(* IEC 61131-3 sources: MyReadCfg/sources/MyReadCfg, 2 files *)

(* ---- MyReadCfg.fun ---- *)
{REDUND_ERROR} FUNCTION MRC_Open : UDINT (*Reads a configuration file into memory, returns Ident (0 = error)*) (*$GROUP=User,$CAT=User,$GROUPICON=User.png,$CATICON=User.png*)
	VAR_INPUT
		pDeviceName : UDINT; (*Pointer to FileIO device name, e.g. 'USER' (STRING)*)
		pFileName : UDINT; (*Pointer to file name incl. relative path, e.g. 'Simulation/50000.INI' (STRING)*)
	END_VAR
END_FUNCTION

{REDUND_ERROR} FUNCTION MRC_Close : DINT (*Closes a configuration and frees all resources. 0 = OK*) (*$GROUP=User,$CAT=User,$GROUPICON=User.png,$CATICON=User.png*)
	VAR_INPUT
		Ident : UDINT; (*Ident from MRC_Open*)
	END_VAR
END_FUNCTION

{REDUND_ERROR} FUNCTION MRC_GetLastError : DINT (*Error of the last MyReadCfg call of this Ident (0 = Ident independent / open error)*) (*$GROUP=User,$CAT=User,$GROUPICON=User.png,$CATICON=User.png*)
	VAR_INPUT
		Ident : UDINT; (*Ident from MRC_Open*)
	END_VAR
END_FUNCTION

{REDUND_ERROR} FUNCTION MRC_KeyExists : BOOL (*TRUE if the key is present*) (*$GROUP=User,$CAT=User,$GROUPICON=User.png,$CATICON=User.png*)
	VAR_INPUT
		Ident : UDINT; (*Ident from MRC_Open*)
		pKey : UDINT; (*pointer to name of the constant (STRING)*)
	END_VAR
END_FUNCTION

{REDUND_ERROR} FUNCTION MRC_ReadBOOL : BOOL (*Reads a value as BOOL*) (*$GROUP=User,$CAT=User,$GROUPICON=User.png,$CATICON=User.png*)
	VAR_INPUT
		Ident : UDINT; (*Ident from MRC_Open*)
		pKey : UDINT; (*Pointer to name of the constant (STRING)*)
		Default : BOOL; (*returned if key is missing or not convertible*)
	END_VAR
END_FUNCTION

{REDUND_ERROR} FUNCTION MRC_ReadDINT : DINT (*Reads a value as DINT*) (*$GROUP=User,$CAT=User,$GROUPICON=User.png,$CATICON=User.png*)
	VAR_INPUT
		Ident : UDINT; (*Ident from MRC_Open*)
		pKey : UDINT; (*Pointer to name of the constant (STRING)*)
		Default : DINT; (*returned if key is missing or not convertible*)
	END_VAR
END_FUNCTION

{REDUND_ERROR} FUNCTION MRC_ReadLREAL : LREAL (*Reads a value as LREAL*) (*$GROUP=User,$CAT=User,$GROUPICON=User.png,$CATICON=User.png*)
	VAR_INPUT
		Ident : UDINT; (*Ident from MRC_Open*)
		pKey : UDINT; (*Pointer to name of the constant (STRING)*)
		Default : LREAL; (*returned if key is missing or not convertible*)
	END_VAR
END_FUNCTION

{REDUND_ERROR} FUNCTION MRC_ReadSTRING : DINT (*Reads a value as STRING. Returns copied length or negative error*) (*$GROUP=User,$CAT=User,$GROUPICON=User.png,$CATICON=User.png*)
	VAR_INPUT
		Ident : UDINT; (*Ident from MRC_Open*)
		pKey : UDINT; (*Pointer to name of the constant (STRING)*)
		pValue : UDINT; (*Pointer to destination buffer (STRING)*)
		MaxSize : UDINT; (*size of destination buffer incl. terminating zero (SIZEOF(STRING))*)
		pDefault : UDINT; (*Pointer to default value, may be 0 (STRING)*)
	END_VAR
END_FUNCTION

{REDUND_ERROR} FUNCTION MRC_ReadContent : DINT (*Reads the complete file content into a STRING variable. Returns copied length or negative error*) (*$GROUP=User,$CAT=User,$GROUPICON=User.png,$CATICON=User.png*)
	VAR_INPUT
		Ident : UDINT; (*Ident from MRC_Open*)
		pValue : UDINT; (*Pointer to destination buffer (STRING)*)
		MaxSize : UDINT; (*size of destination buffer incl. terminating zero (SIZEOF(STRING))*)
	END_VAR
END_FUNCTION

(* ---- MyReadCfgConstants.var ---- *)
VAR CONSTANT
	MRC_MAX_HANDLES : UDINT := 8; (*number of configurations that can be open at the same time*)
	MRC_MAX_FILE_SIZE : UDINT := 1048576; (*1 MiB*)
	MRC_MAX_KEY_LENGTH : UDINT := 64;
	MRC_MAX_VALUE_LENGTH : UDINT := 255;
	MRC_READ_CHUNK : UDINT := 8192; (*block size for FileRead*)
	MRC_FILEIO_MAX_CALLS : UDINT := 100000; (*loop guard for asynchronous function blocks*)
	MRC_LOGGER_SIZE : UDINT := 65536; (*size of the logger in bytes, fixed at creation*)

	MRC_EVENT_INFO : DINT := 1610612736;
	MRC_EVENT_WARN : DINT := -1610612736;
	MRC_EVENT_ERR : DINT := -536870912;

	MRC_ERR_OK : DINT := 0;
	MRC_ERR_PARAM : DINT := -1064370176; (*invalid parameter*)
	MRC_ERR_INVALID_IDENT : DINT := -1064370175; (*unknown or closed Ident*)
	MRC_ERR_NO_HANDLE : DINT := -1064370174; (*handle table full*)
	MRC_ERR_FILE : DINT := -1064370173; (*FileIO error*)
	MRC_ERR_FILE_TOO_BIG : DINT := -1064370172;
	MRC_ERR_MEMORY : DINT := -1064370171;
	MRC_ERR_KEY_NOT_FOUND : DINT := -1064370170;
	MRC_ERR_CONVERSION : DINT := -1064370169;
	MRC_ERR_TRUNCATED : DINT := -1064370168;
	MRC_ERR_TIMEOUT : DINT := -1064370167; (*asynchronous function block did not finish*)
END_VAR
